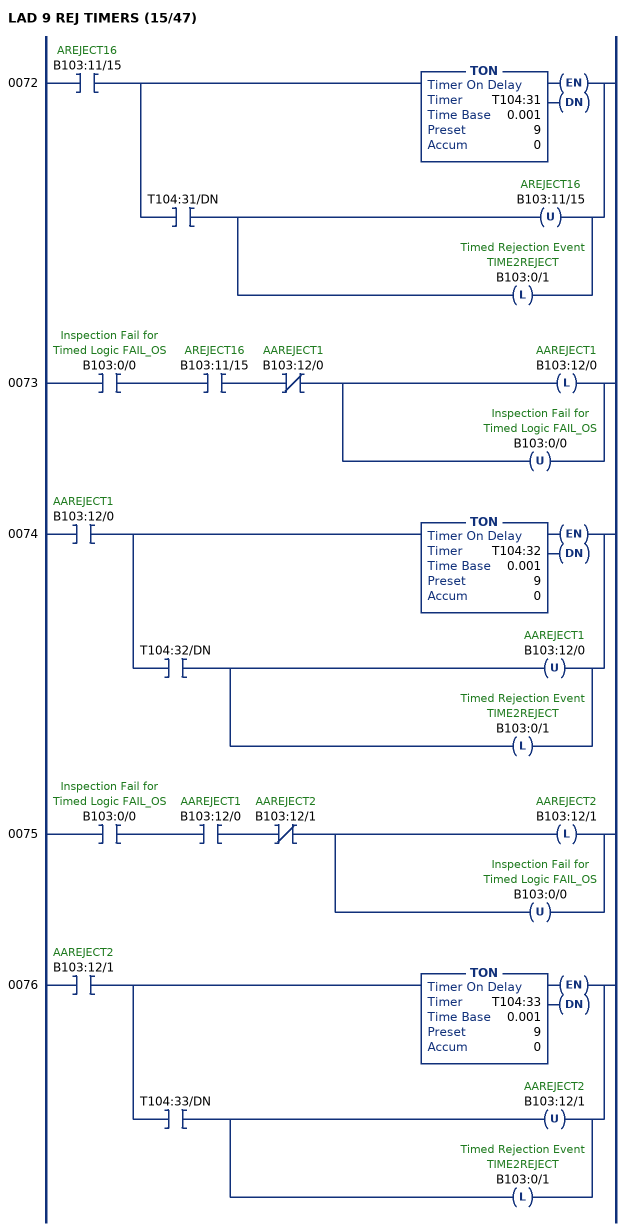
% Rung: 72 %
SOR XIC B103:11/15 BST TON T104:31 0.001 9 0 NXB XIC T104:31/DN BST OTU B103:11/15 NXB OTL B103:0/1 BND BND EOR
%   B103:11/15  AREJECT16 %
%   B103:0/1  TIME2REJECT  "Timed Rejection Event" %
% Rung: 73 %
SOR XIC B103:0/0 XIC B103:11/15 XIO B103:12/0 BST OTL B103:12/0 NXB OTU B103:0/0 BND EOR
%   B103:0/0  FAIL_OS  "Inspection Fail for Timed Logic" %
%   B103:11/15  AREJECT16 %
%   B103:12/0  AAREJECT1 %
% Rung: 74 %
SOR XIC B103:12/0 BST TON T104:32 0.001 9 0 NXB XIC T104:32/DN BST OTU B103:12/0 NXB OTL B103:0/1 BND BND EOR
%   B103:12/0  AAREJECT1 %
%   B103:0/1  TIME2REJECT  "Timed Rejection Event" %
% Rung: 75 %
SOR XIC B103:0/0 XIC B103:12/0 XIO B103:12/1 BST OTL B103:12/1 NXB OTU B103:0/0 BND EOR
%   B103:0/0  FAIL_OS  "Inspection Fail for Timed Logic" %
%   B103:12/0  AAREJECT1 %
%   B103:12/1  AAREJECT2 %
% Rung: 76 %
SOR XIC B103:12/1 BST TON T104:33 0.001 9 0 NXB XIC T104:33/DN BST OTU B103:12/1 NXB OTL B103:0/1 BND BND EOR
%   B103:12/1  AAREJECT2 %
%   B103:0/1  TIME2REJECT  "Timed Rejection Event" %

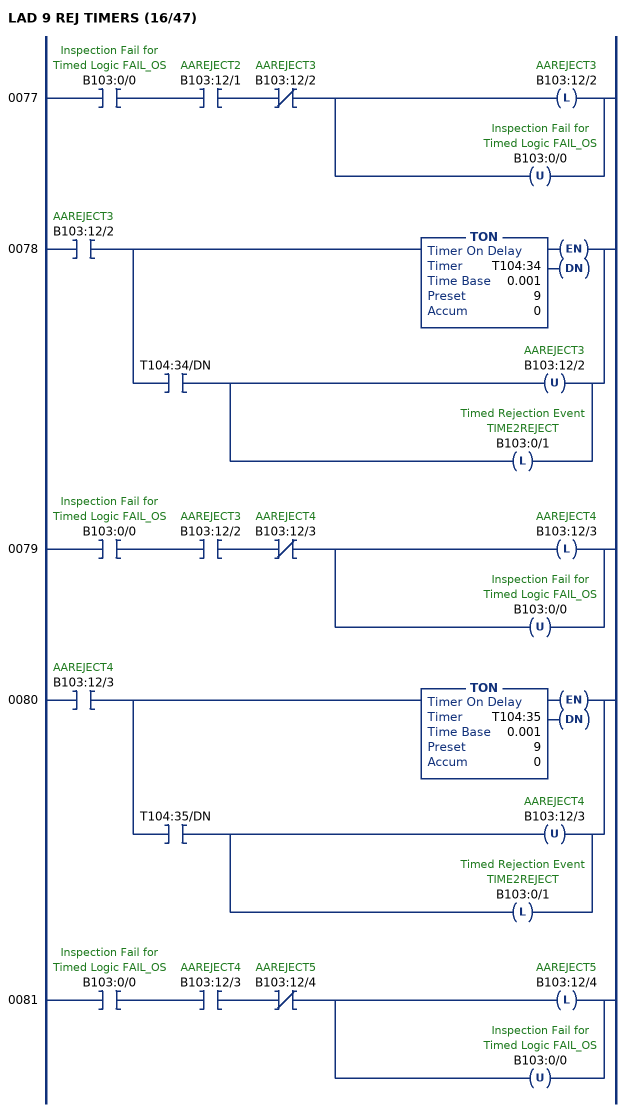
% Rung: 77 %
SOR XIC B103:0/0 XIC B103:12/1 XIO B103:12/2 BST OTL B103:12/2 NXB OTU B103:0/0 BND EOR
%   B103:0/0  FAIL_OS  "Inspection Fail for Timed Logic" %
%   B103:12/1  AAREJECT2 %
%   B103:12/2  AAREJECT3 %
% Rung: 78 %
SOR XIC B103:12/2 BST TON T104:34 0.001 9 0 NXB XIC T104:34/DN BST OTU B103:12/2 NXB OTL B103:0/1 BND BND EOR
%   B103:12/2  AAREJECT3 %
%   B103:0/1  TIME2REJECT  "Timed Rejection Event" %
% Rung: 79 %
SOR XIC B103:0/0 XIC B103:12/2 XIO B103:12/3 BST OTL B103:12/3 NXB OTU B103:0/0 BND EOR
%   B103:0/0  FAIL_OS  "Inspection Fail for Timed Logic" %
%   B103:12/2  AAREJECT3 %
%   B103:12/3  AAREJECT4 %
% Rung: 80 %
SOR XIC B103:12/3 BST TON T104:35 0.001 9 0 NXB XIC T104:35/DN BST OTU B103:12/3 NXB OTL B103:0/1 BND BND EOR
%   B103:12/3  AAREJECT4 %
%   B103:0/1  TIME2REJECT  "Timed Rejection Event" %
% Rung: 81 %
SOR XIC B103:0/0 XIC B103:12/3 XIO B103:12/4 BST OTL B103:12/4 NXB OTU B103:0/0 BND EOR
%   B103:0/0  FAIL_OS  "Inspection Fail for Timed Logic" %
%   B103:12/3  AAREJECT4 %
%   B103:12/4  AAREJECT5 %

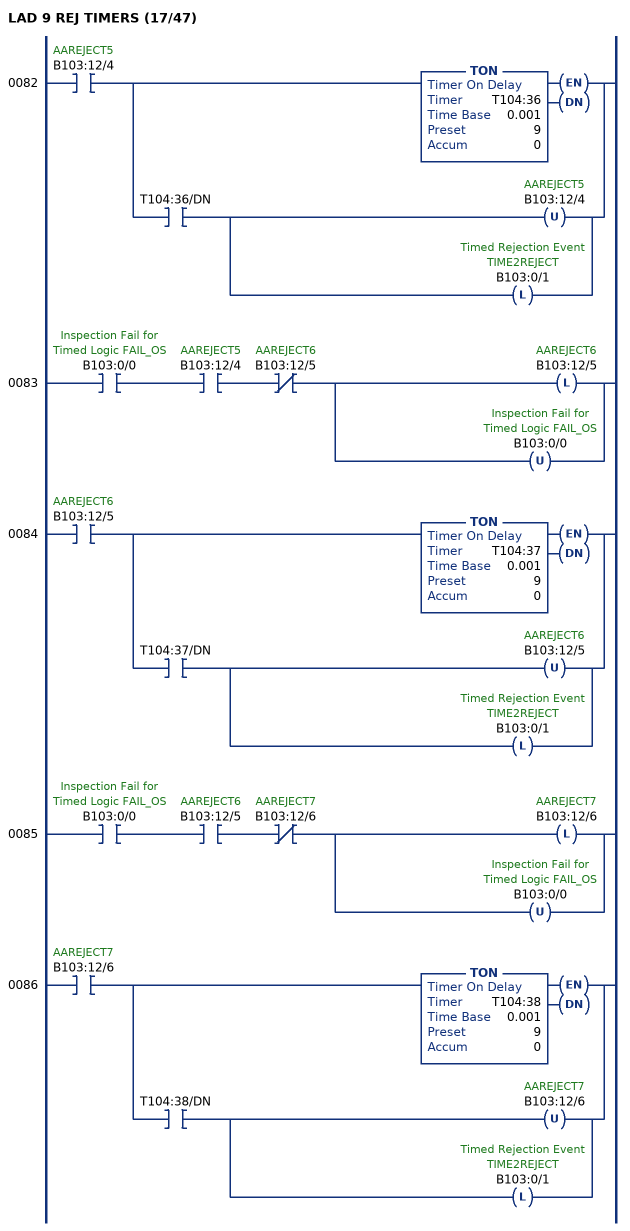
% Rung: 82 %
SOR XIC B103:12/4 BST TON T104:36 0.001 9 0 NXB XIC T104:36/DN BST OTU B103:12/4 NXB OTL B103:0/1 BND BND EOR
%   B103:12/4  AAREJECT5 %
%   B103:0/1  TIME2REJECT  "Timed Rejection Event" %
% Rung: 83 %
SOR XIC B103:0/0 XIC B103:12/4 XIO B103:12/5 BST OTL B103:12/5 NXB OTU B103:0/0 BND EOR
%   B103:0/0  FAIL_OS  "Inspection Fail for Timed Logic" %
%   B103:12/4  AAREJECT5 %
%   B103:12/5  AAREJECT6 %
% Rung: 84 %
SOR XIC B103:12/5 BST TON T104:37 0.001 9 0 NXB XIC T104:37/DN BST OTU B103:12/5 NXB OTL B103:0/1 BND BND EOR
%   B103:12/5  AAREJECT6 %
%   B103:0/1  TIME2REJECT  "Timed Rejection Event" %
% Rung: 85 %
SOR XIC B103:0/0 XIC B103:12/5 XIO B103:12/6 BST OTL B103:12/6 NXB OTU B103:0/0 BND EOR
%   B103:0/0  FAIL_OS  "Inspection Fail for Timed Logic" %
%   B103:12/5  AAREJECT6 %
%   B103:12/6  AAREJECT7 %
% Rung: 86 %
SOR XIC B103:12/6 BST TON T104:38 0.001 9 0 NXB XIC T104:38/DN BST OTU B103:12/6 NXB OTL B103:0/1 BND BND EOR
%   B103:12/6  AAREJECT7 %
%   B103:0/1  TIME2REJECT  "Timed Rejection Event" %

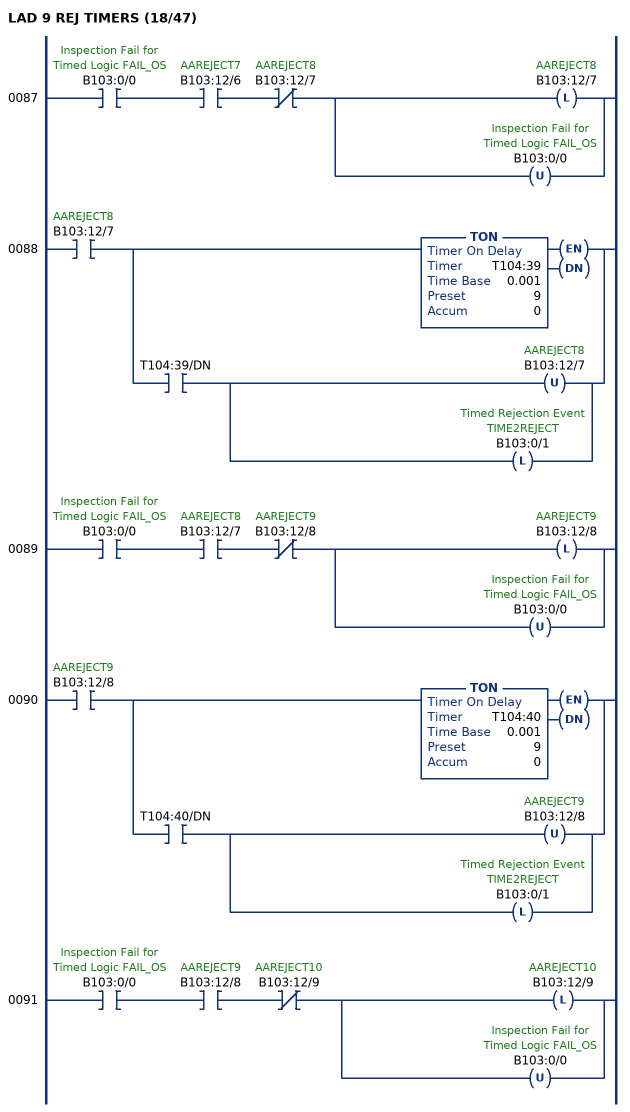
% Rung: 87 %
SOR XIC B103:0/0 XIC B103:12/6 XIO B103:12/7 BST OTL B103:12/7 NXB OTU B103:0/0 BND EOR
%   B103:0/0  FAIL_OS  "Inspection Fail for Timed Logic" %
%   B103:12/6  AAREJECT7 %
%   B103:12/7  AAREJECT8 %
% Rung: 88 %
SOR XIC B103:12/7 BST TON T104:39 0.001 9 0 NXB XIC T104:39/DN BST OTU B103:12/7 NXB OTL B103:0/1 BND BND EOR
%   B103:12/7  AAREJECT8 %
%   B103:0/1  TIME2REJECT  "Timed Rejection Event" %
% Rung: 89 %
SOR XIC B103:0/0 XIC B103:12/7 XIO B103:12/8 BST OTL B103:12/8 NXB OTU B103:0/0 BND EOR
%   B103:0/0  FAIL_OS  "Inspection Fail for Timed Logic" %
%   B103:12/7  AAREJECT8 %
%   B103:12/8  AAREJECT9 %
% Rung: 90 %
SOR XIC B103:12/8 BST TON T104:40 0.001 9 0 NXB XIC T104:40/DN BST OTU B103:12/8 NXB OTL B103:0/1 BND BND EOR
%   B103:12/8  AAREJECT9 %
%   B103:0/1  TIME2REJECT  "Timed Rejection Event" %
% Rung: 91 %
SOR XIC B103:0/0 XIC B103:12/8 XIO B103:12/9 BST OTL B103:12/9 NXB OTU B103:0/0 BND EOR
%   B103:0/0  FAIL_OS  "Inspection Fail for Timed Logic" %
%   B103:12/8  AAREJECT9 %
%   B103:12/9  AAREJECT10 %

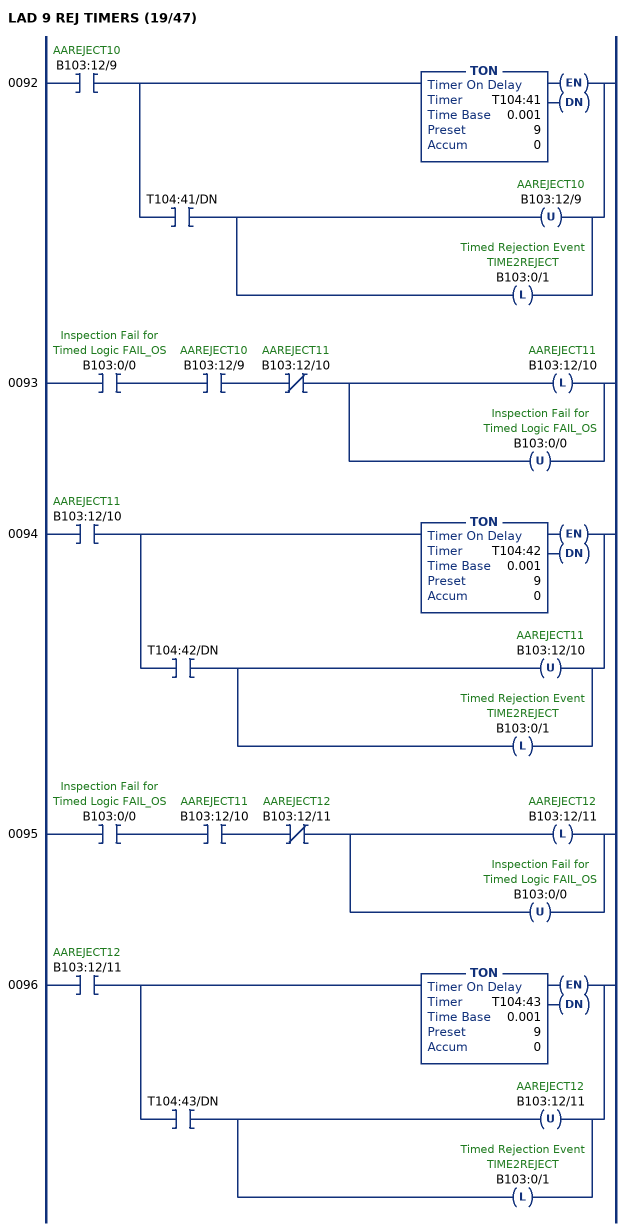
% Rung: 92 %
SOR XIC B103:12/9 BST TON T104:41 0.001 9 0 NXB XIC T104:41/DN BST OTU B103:12/9 NXB OTL B103:0/1 BND BND EOR
%   B103:12/9  AAREJECT10 %
%   B103:0/1  TIME2REJECT  "Timed Rejection Event" %
% Rung: 93 %
SOR XIC B103:0/0 XIC B103:12/9 XIO B103:12/10 BST OTL B103:12/10 NXB OTU B103:0/0 BND EOR
%   B103:0/0  FAIL_OS  "Inspection Fail for Timed Logic" %
%   B103:12/9  AAREJECT10 %
%   B103:12/10  AAREJECT11 %
% Rung: 94 %
SOR XIC B103:12/10 BST TON T104:42 0.001 9 0 NXB XIC T104:42/DN BST OTU B103:12/10 NXB OTL B103:0/1 BND BND EOR
%   B103:12/10  AAREJECT11 %
%   B103:0/1  TIME2REJECT  "Timed Rejection Event" %
% Rung: 95 %
SOR XIC B103:0/0 XIC B103:12/10 XIO B103:12/11 BST OTL B103:12/11 NXB OTU B103:0/0 BND EOR
%   B103:0/0  FAIL_OS  "Inspection Fail for Timed Logic" %
%   B103:12/10  AAREJECT11 %
%   B103:12/11  AAREJECT12 %
% Rung: 96 %
SOR XIC B103:12/11 BST TON T104:43 0.001 9 0 NXB XIC T104:43/DN BST OTU B103:12/11 NXB OTL B103:0/1 BND BND EOR
%   B103:12/11  AAREJECT12 %
%   B103:0/1  TIME2REJECT  "Timed Rejection Event" %

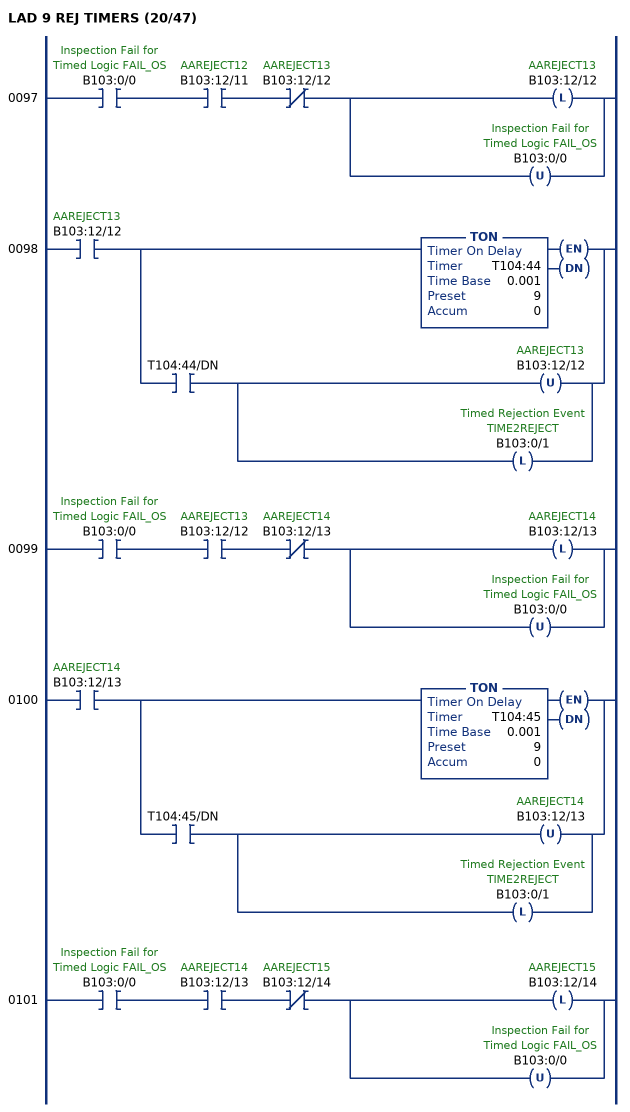
% Rung: 97 %
SOR XIC B103:0/0 XIC B103:12/11 XIO B103:12/12 BST OTL B103:12/12 NXB OTU B103:0/0 BND EOR
%   B103:0/0  FAIL_OS  "Inspection Fail for Timed Logic" %
%   B103:12/11  AAREJECT12 %
%   B103:12/12  AAREJECT13 %
% Rung: 98 %
SOR XIC B103:12/12 BST TON T104:44 0.001 9 0 NXB XIC T104:44/DN BST OTU B103:12/12 NXB OTL B103:0/1 BND BND EOR
%   B103:12/12  AAREJECT13 %
%   B103:0/1  TIME2REJECT  "Timed Rejection Event" %
% Rung: 99 %
SOR XIC B103:0/0 XIC B103:12/12 XIO B103:12/13 BST OTL B103:12/13 NXB OTU B103:0/0 BND EOR
%   B103:0/0  FAIL_OS  "Inspection Fail for Timed Logic" %
%   B103:12/12  AAREJECT13 %
%   B103:12/13  AAREJECT14 %
% Rung: 100 %
SOR XIC B103:12/13 BST TON T104:45 0.001 9 0 NXB XIC T104:45/DN BST OTU B103:12/13 NXB OTL B103:0/1 BND BND EOR
%   B103:12/13  AAREJECT14 %
%   B103:0/1  TIME2REJECT  "Timed Rejection Event" %
% Rung: 101 %
SOR XIC B103:0/0 XIC B103:12/13 XIO B103:12/14 BST OTL B103:12/14 NXB OTU B103:0/0 BND EOR
%   B103:0/0  FAIL_OS  "Inspection Fail for Timed Logic" %
%   B103:12/13  AAREJECT14 %
%   B103:12/14  AAREJECT15 %

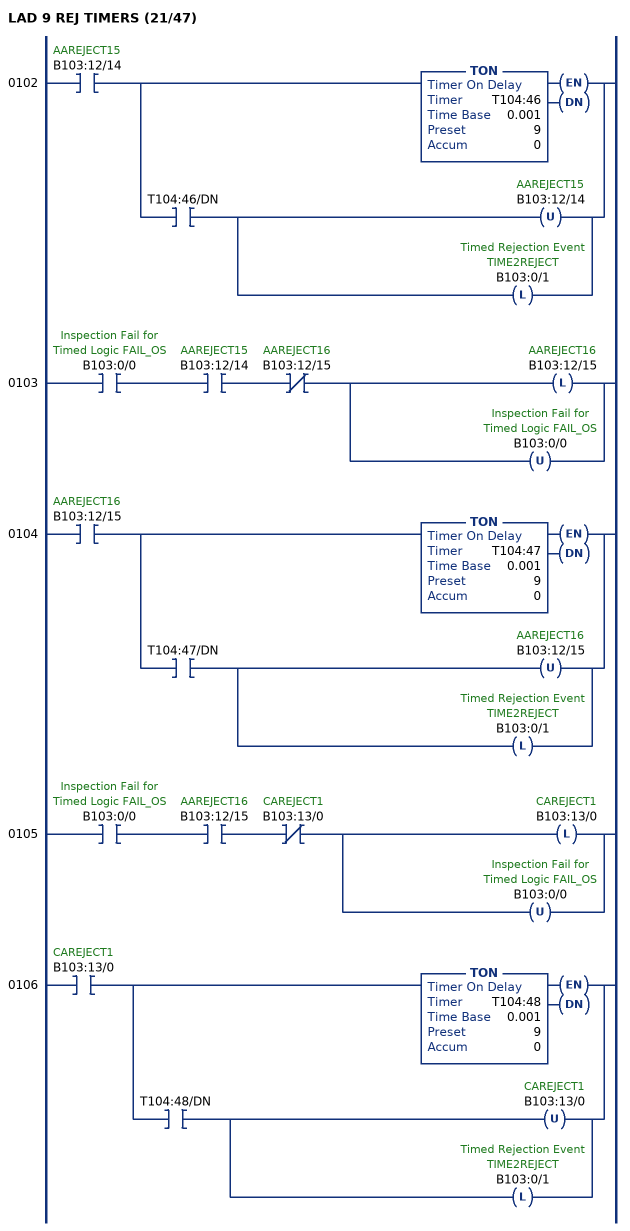
% Rung: 102 %
SOR XIC B103:12/14 BST TON T104:46 0.001 9 0 NXB XIC T104:46/DN BST OTU B103:12/14 NXB OTL B103:0/1 BND BND EOR
%   B103:12/14  AAREJECT15 %
%   B103:0/1  TIME2REJECT  "Timed Rejection Event" %
% Rung: 103 %
SOR XIC B103:0/0 XIC B103:12/14 XIO B103:12/15 BST OTL B103:12/15 NXB OTU B103:0/0 BND EOR
%   B103:0/0  FAIL_OS  "Inspection Fail for Timed Logic" %
%   B103:12/14  AAREJECT15 %
%   B103:12/15  AAREJECT16 %
% Rung: 104 %
SOR XIC B103:12/15 BST TON T104:47 0.001 9 0 NXB XIC T104:47/DN BST OTU B103:12/15 NXB OTL B103:0/1 BND BND EOR
%   B103:12/15  AAREJECT16 %
%   B103:0/1  TIME2REJECT  "Timed Rejection Event" %
% Rung: 105 %
SOR XIC B103:0/0 XIC B103:12/15 XIO B103:13/0 BST OTL B103:13/0 NXB OTU B103:0/0 BND EOR
%   B103:0/0  FAIL_OS  "Inspection Fail for Timed Logic" %
%   B103:12/15  AAREJECT16 %
%   B103:13/0  CAREJECT1 %
% Rung: 106 %
SOR XIC B103:13/0 BST TON T104:48 0.001 9 0 NXB XIC T104:48/DN BST OTU B103:13/0 NXB OTL B103:0/1 BND BND EOR
%   B103:13/0  CAREJECT1 %
%   B103:0/1  TIME2REJECT  "Timed Rejection Event" %

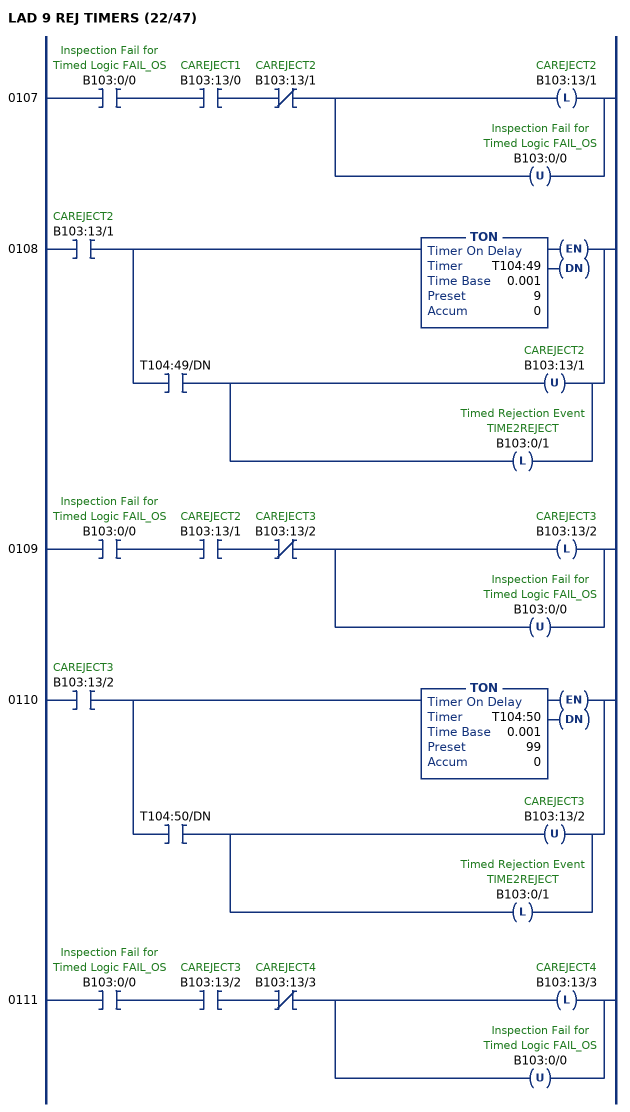
% Rung: 107 %
SOR XIC B103:0/0 XIC B103:13/0 XIO B103:13/1 BST OTL B103:13/1 NXB OTU B103:0/0 BND EOR
%   B103:0/0  FAIL_OS  "Inspection Fail for Timed Logic" %
%   B103:13/0  CAREJECT1 %
%   B103:13/1  CAREJECT2 %
% Rung: 108 %
SOR XIC B103:13/1 BST TON T104:49 0.001 9 0 NXB XIC T104:49/DN BST OTU B103:13/1 NXB OTL B103:0/1 BND BND EOR
%   B103:13/1  CAREJECT2 %
%   B103:0/1  TIME2REJECT  "Timed Rejection Event" %
% Rung: 109 %
SOR XIC B103:0/0 XIC B103:13/1 XIO B103:13/2 BST OTL B103:13/2 NXB OTU B103:0/0 BND EOR
%   B103:0/0  FAIL_OS  "Inspection Fail for Timed Logic" %
%   B103:13/1  CAREJECT2 %
%   B103:13/2  CAREJECT3 %
% Rung: 110 %
SOR XIC B103:13/2 BST TON T104:50 0.001 99 0 NXB XIC T104:50/DN BST OTU B103:13/2 NXB OTL B103:0/1 BND BND EOR
%   B103:13/2  CAREJECT3 %
%   B103:0/1  TIME2REJECT  "Timed Rejection Event" %
% Rung: 111 %
SOR XIC B103:0/0 XIC B103:13/2 XIO B103:13/3 BST OTL B103:13/3 NXB OTU B103:0/0 BND EOR
%   B103:0/0  FAIL_OS  "Inspection Fail for Timed Logic" %
%   B103:13/2  CAREJECT3 %
%   B103:13/3  CAREJECT4 %

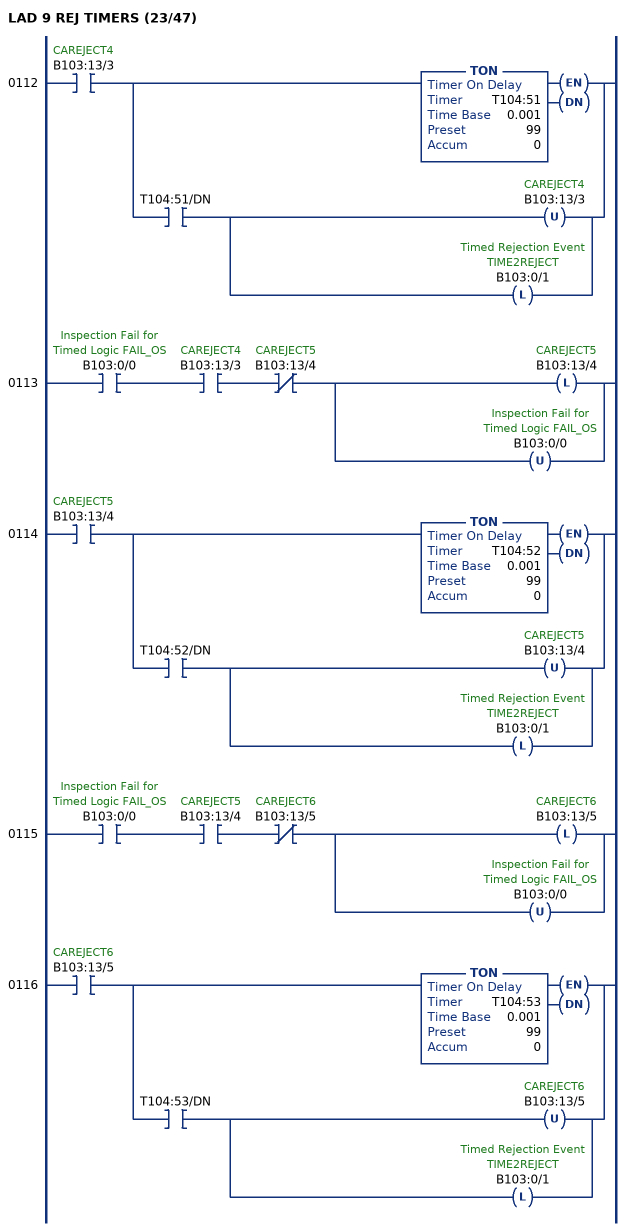
% Rung: 112 %
SOR XIC B103:13/3 BST TON T104:51 0.001 99 0 NXB XIC T104:51/DN BST OTU B103:13/3 NXB OTL B103:0/1 BND BND EOR
%   B103:13/3  CAREJECT4 %
%   B103:0/1  TIME2REJECT  "Timed Rejection Event" %
% Rung: 113 %
SOR XIC B103:0/0 XIC B103:13/3 XIO B103:13/4 BST OTL B103:13/4 NXB OTU B103:0/0 BND EOR
%   B103:0/0  FAIL_OS  "Inspection Fail for Timed Logic" %
%   B103:13/3  CAREJECT4 %
%   B103:13/4  CAREJECT5 %
% Rung: 114 %
SOR XIC B103:13/4 BST TON T104:52 0.001 99 0 NXB XIC T104:52/DN BST OTU B103:13/4 NXB OTL B103:0/1 BND BND EOR
%   B103:13/4  CAREJECT5 %
%   B103:0/1  TIME2REJECT  "Timed Rejection Event" %
% Rung: 115 %
SOR XIC B103:0/0 XIC B103:13/4 XIO B103:13/5 BST OTL B103:13/5 NXB OTU B103:0/0 BND EOR
%   B103:0/0  FAIL_OS  "Inspection Fail for Timed Logic" %
%   B103:13/4  CAREJECT5 %
%   B103:13/5  CAREJECT6 %
% Rung: 116 %
SOR XIC B103:13/5 BST TON T104:53 0.001 99 0 NXB XIC T104:53/DN BST OTU B103:13/5 NXB OTL B103:0/1 BND BND EOR
%   B103:13/5  CAREJECT6 %
%   B103:0/1  TIME2REJECT  "Timed Rejection Event" %

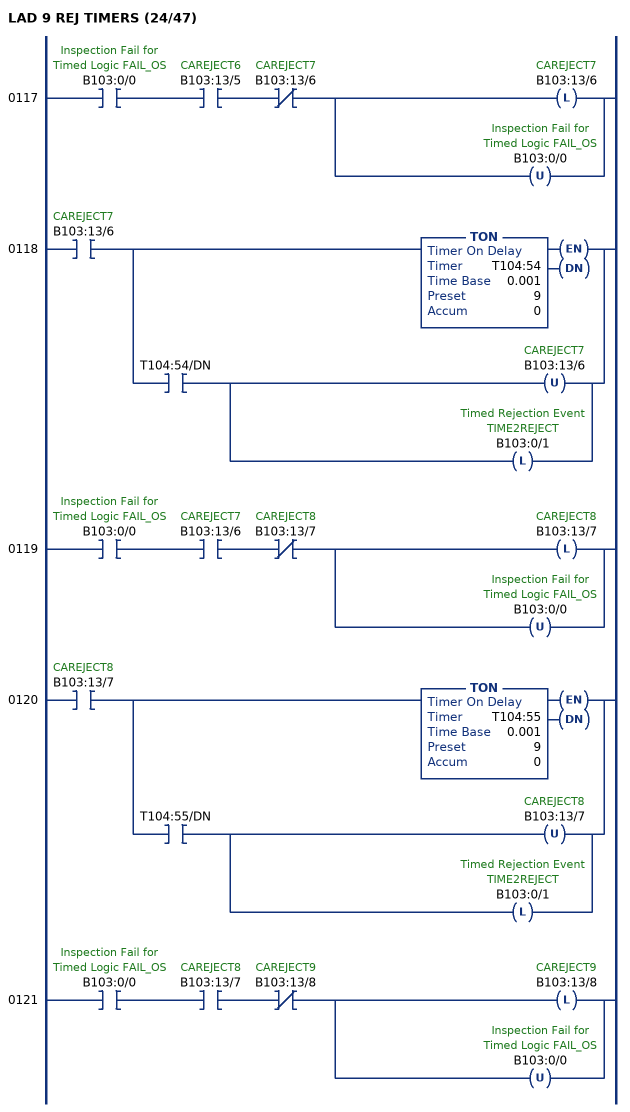
% Rung: 117 %
SOR XIC B103:0/0 XIC B103:13/5 XIO B103:13/6 BST OTL B103:13/6 NXB OTU B103:0/0 BND EOR
%   B103:0/0  FAIL_OS  "Inspection Fail for Timed Logic" %
%   B103:13/5  CAREJECT6 %
%   B103:13/6  CAREJECT7 %
% Rung: 118 %
SOR XIC B103:13/6 BST TON T104:54 0.001 9 0 NXB XIC T104:54/DN BST OTU B103:13/6 NXB OTL B103:0/1 BND BND EOR
%   B103:13/6  CAREJECT7 %
%   B103:0/1  TIME2REJECT  "Timed Rejection Event" %
% Rung: 119 %
SOR XIC B103:0/0 XIC B103:13/6 XIO B103:13/7 BST OTL B103:13/7 NXB OTU B103:0/0 BND EOR
%   B103:0/0  FAIL_OS  "Inspection Fail for Timed Logic" %
%   B103:13/6  CAREJECT7 %
%   B103:13/7  CAREJECT8 %
% Rung: 120 %
SOR XIC B103:13/7 BST TON T104:55 0.001 9 0 NXB XIC T104:55/DN BST OTU B103:13/7 NXB OTL B103:0/1 BND BND EOR
%   B103:13/7  CAREJECT8 %
%   B103:0/1  TIME2REJECT  "Timed Rejection Event" %
% Rung: 121 %
SOR XIC B103:0/0 XIC B103:13/7 XIO B103:13/8 BST OTL B103:13/8 NXB OTU B103:0/0 BND EOR
%   B103:0/0  FAIL_OS  "Inspection Fail for Timed Logic" %
%   B103:13/7  CAREJECT8 %
%   B103:13/8  CAREJECT9 %

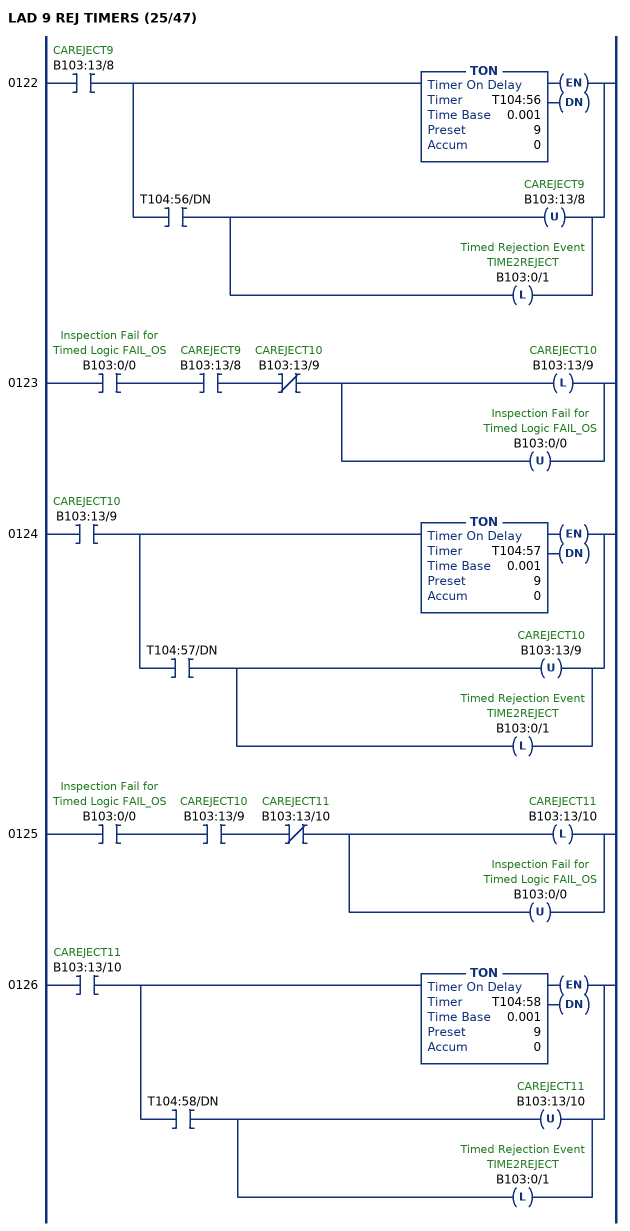
% Rung: 122 %
SOR XIC B103:13/8 BST TON T104:56 0.001 9 0 NXB XIC T104:56/DN BST OTU B103:13/8 NXB OTL B103:0/1 BND BND EOR
%   B103:13/8  CAREJECT9 %
%   B103:0/1  TIME2REJECT  "Timed Rejection Event" %
% Rung: 123 %
SOR XIC B103:0/0 XIC B103:13/8 XIO B103:13/9 BST OTL B103:13/9 NXB OTU B103:0/0 BND EOR
%   B103:0/0  FAIL_OS  "Inspection Fail for Timed Logic" %
%   B103:13/8  CAREJECT9 %
%   B103:13/9  CAREJECT10 %
% Rung: 124 %
SOR XIC B103:13/9 BST TON T104:57 0.001 9 0 NXB XIC T104:57/DN BST OTU B103:13/9 NXB OTL B103:0/1 BND BND EOR
%   B103:13/9  CAREJECT10 %
%   B103:0/1  TIME2REJECT  "Timed Rejection Event" %
% Rung: 125 %
SOR XIC B103:0/0 XIC B103:13/9 XIO B103:13/10 BST OTL B103:13/10 NXB OTU B103:0/0 BND EOR
%   B103:0/0  FAIL_OS  "Inspection Fail for Timed Logic" %
%   B103:13/9  CAREJECT10 %
%   B103:13/10  CAREJECT11 %
% Rung: 126 %
SOR XIC B103:13/10 BST TON T104:58 0.001 9 0 NXB XIC T104:58/DN BST OTU B103:13/10 NXB OTL B103:0/1 BND BND EOR
%   B103:13/10  CAREJECT11 %
%   B103:0/1  TIME2REJECT  "Timed Rejection Event" %

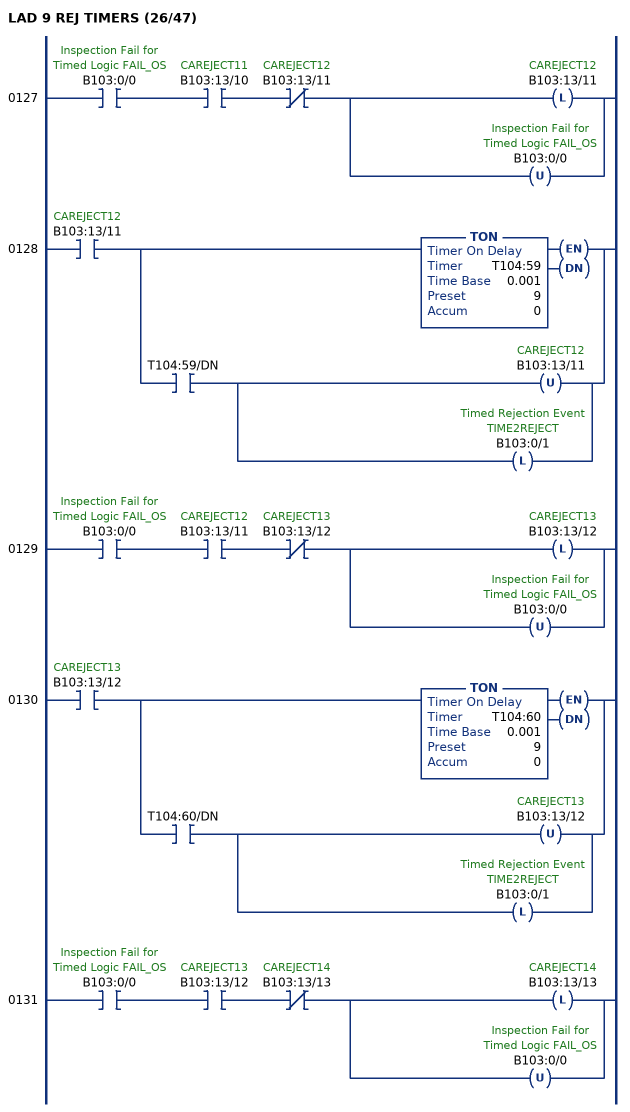
% Rung: 127 %
SOR XIC B103:0/0 XIC B103:13/10 XIO B103:13/11 BST OTL B103:13/11 NXB OTU B103:0/0 BND EOR
%   B103:0/0  FAIL_OS  "Inspection Fail for Timed Logic" %
%   B103:13/10  CAREJECT11 %
%   B103:13/11  CAREJECT12 %
% Rung: 128 %
SOR XIC B103:13/11 BST TON T104:59 0.001 9 0 NXB XIC T104:59/DN BST OTU B103:13/11 NXB OTL B103:0/1 BND BND EOR
%   B103:13/11  CAREJECT12 %
%   B103:0/1  TIME2REJECT  "Timed Rejection Event" %
% Rung: 129 %
SOR XIC B103:0/0 XIC B103:13/11 XIO B103:13/12 BST OTL B103:13/12 NXB OTU B103:0/0 BND EOR
%   B103:0/0  FAIL_OS  "Inspection Fail for Timed Logic" %
%   B103:13/11  CAREJECT12 %
%   B103:13/12  CAREJECT13 %
% Rung: 130 %
SOR XIC B103:13/12 BST TON T104:60 0.001 9 0 NXB XIC T104:60/DN BST OTU B103:13/12 NXB OTL B103:0/1 BND BND EOR
%   B103:13/12  CAREJECT13 %
%   B103:0/1  TIME2REJECT  "Timed Rejection Event" %
% Rung: 131 %
SOR XIC B103:0/0 XIC B103:13/12 XIO B103:13/13 BST OTL B103:13/13 NXB OTU B103:0/0 BND EOR
%   B103:0/0  FAIL_OS  "Inspection Fail for Timed Logic" %
%   B103:13/12  CAREJECT13 %
%   B103:13/13  CAREJECT14 %

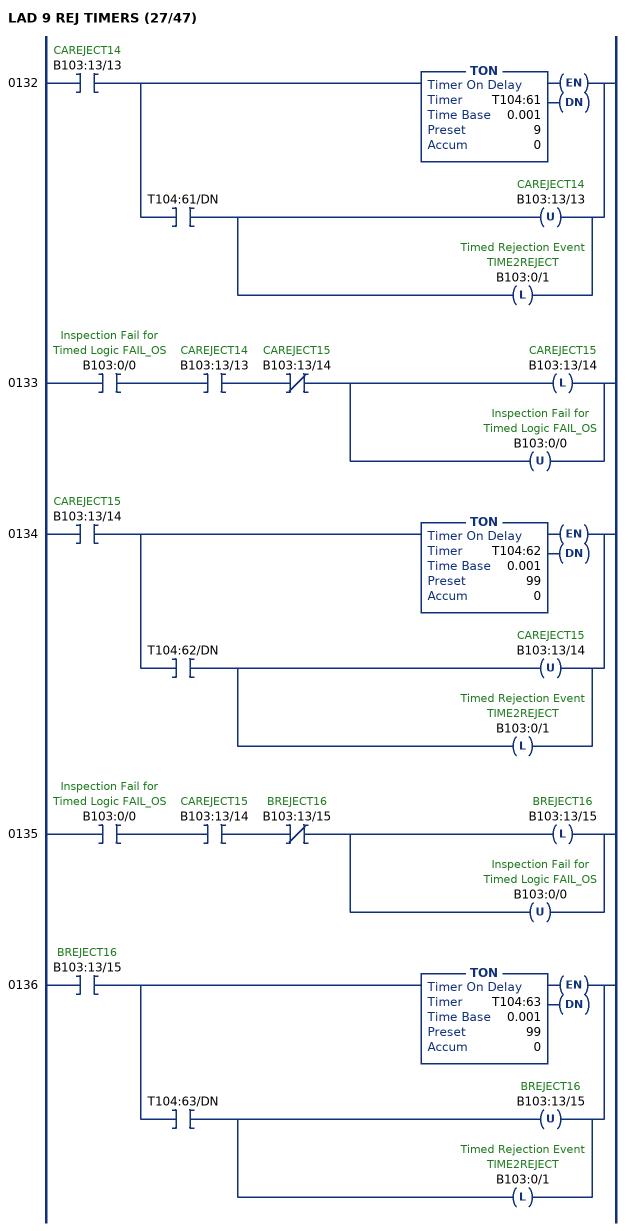
% Rung: 132 %
SOR XIC B103:13/13 BST TON T104:61 0.001 9 0 NXB XIC T104:61/DN BST OTU B103:13/13 NXB OTL B103:0/1 BND BND EOR
%   B103:13/13  CAREJECT14 %
%   B103:0/1  TIME2REJECT  "Timed Rejection Event" %
% Rung: 133 %
SOR XIC B103:0/0 XIC B103:13/13 XIO B103:13/14 BST OTL B103:13/14 NXB OTU B103:0/0 BND EOR
%   B103:0/0  FAIL_OS  "Inspection Fail for Timed Logic" %
%   B103:13/13  CAREJECT14 %
%   B103:13/14  CAREJECT15 %
% Rung: 134 %
SOR XIC B103:13/14 BST TON T104:62 0.001 99 0 NXB XIC T104:62/DN BST OTU B103:13/14 NXB OTL B103:0/1 BND BND EOR
%   B103:13/14  CAREJECT15 %
%   B103:0/1  TIME2REJECT  "Timed Rejection Event" %
% Rung: 135 %
SOR XIC B103:0/0 XIC B103:13/14 XIO B103:13/15 BST OTL B103:13/15 NXB OTU B103:0/0 BND EOR
%   B103:0/0  FAIL_OS  "Inspection Fail for Timed Logic" %
%   B103:13/14  CAREJECT15 %
%   B103:13/15  BREJECT16 %
% Rung: 136 %
SOR XIC B103:13/15 BST TON T104:63 0.001 99 0 NXB XIC T104:63/DN BST OTU B103:13/15 NXB OTL B103:0/1 BND BND EOR
%   B103:13/15  BREJECT16 %
%   B103:0/1  TIME2REJECT  "Timed Rejection Event" %

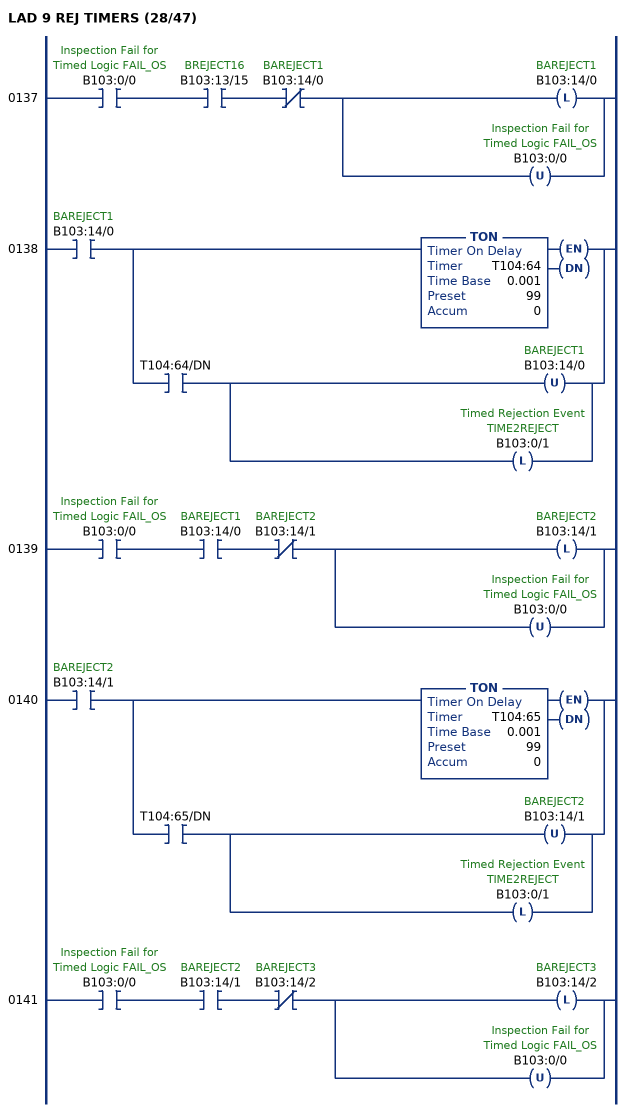
% Rung: 137 %
SOR XIC B103:0/0 XIC B103:13/15 XIO B103:14/0 BST OTL B103:14/0 NXB OTU B103:0/0 BND EOR
%   B103:0/0  FAIL_OS  "Inspection Fail for Timed Logic" %
%   B103:13/15  BREJECT16 %
%   B103:14/0  BAREJECT1 %
% Rung: 138 %
SOR XIC B103:14/0 BST TON T104:64 0.001 99 0 NXB XIC T104:64/DN BST OTU B103:14/0 NXB OTL B103:0/1 BND BND EOR
%   B103:14/0  BAREJECT1 %
%   B103:0/1  TIME2REJECT  "Timed Rejection Event" %
% Rung: 139 %
SOR XIC B103:0/0 XIC B103:14/0 XIO B103:14/1 BST OTL B103:14/1 NXB OTU B103:0/0 BND EOR
%   B103:0/0  FAIL_OS  "Inspection Fail for Timed Logic" %
%   B103:14/0  BAREJECT1 %
%   B103:14/1  BAREJECT2 %
% Rung: 140 %
SOR XIC B103:14/1 BST TON T104:65 0.001 99 0 NXB XIC T104:65/DN BST OTU B103:14/1 NXB OTL B103:0/1 BND BND EOR
%   B103:14/1  BAREJECT2 %
%   B103:0/1  TIME2REJECT  "Timed Rejection Event" %
% Rung: 141 %
SOR XIC B103:0/0 XIC B103:14/1 XIO B103:14/2 BST OTL B103:14/2 NXB OTU B103:0/0 BND EOR
%   B103:0/0  FAIL_OS  "Inspection Fail for Timed Logic" %
%   B103:14/1  BAREJECT2 %
%   B103:14/2  BAREJECT3 %

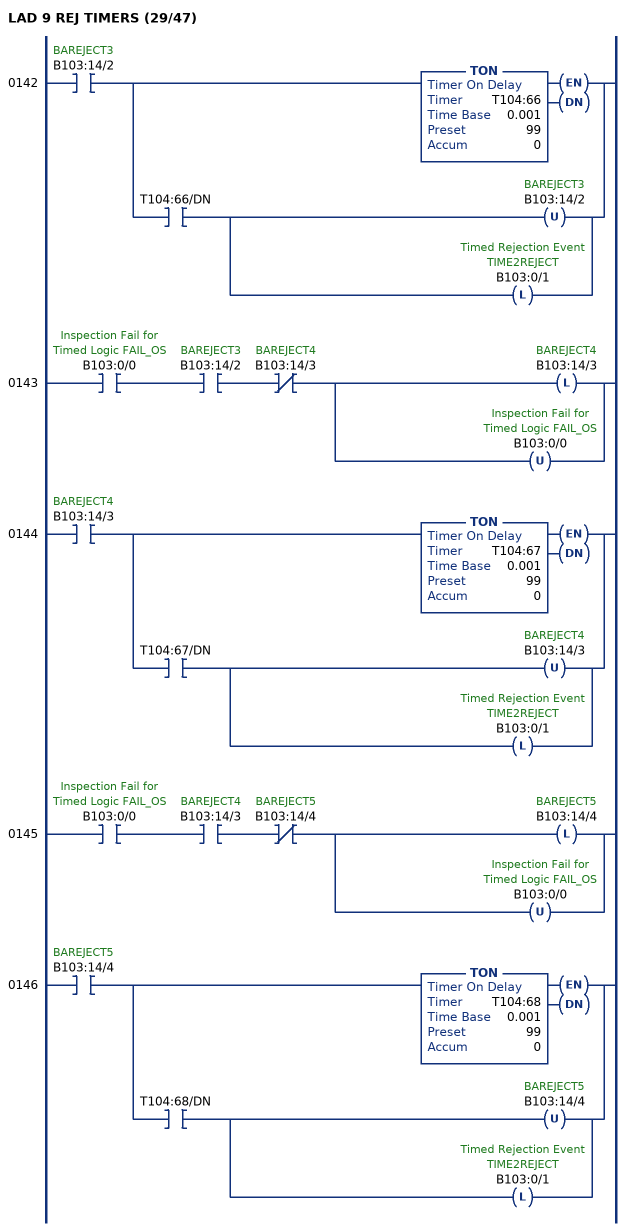
% Rung: 142 %
SOR XIC B103:14/2 BST TON T104:66 0.001 99 0 NXB XIC T104:66/DN BST OTU B103:14/2 NXB OTL B103:0/1 BND BND EOR
%   B103:14/2  BAREJECT3 %
%   B103:0/1  TIME2REJECT  "Timed Rejection Event" %
% Rung: 143 %
SOR XIC B103:0/0 XIC B103:14/2 XIO B103:14/3 BST OTL B103:14/3 NXB OTU B103:0/0 BND EOR
%   B103:0/0  FAIL_OS  "Inspection Fail for Timed Logic" %
%   B103:14/2  BAREJECT3 %
%   B103:14/3  BAREJECT4 %
% Rung: 144 %
SOR XIC B103:14/3 BST TON T104:67 0.001 99 0 NXB XIC T104:67/DN BST OTU B103:14/3 NXB OTL B103:0/1 BND BND EOR
%   B103:14/3  BAREJECT4 %
%   B103:0/1  TIME2REJECT  "Timed Rejection Event" %
% Rung: 145 %
SOR XIC B103:0/0 XIC B103:14/3 XIO B103:14/4 BST OTL B103:14/4 NXB OTU B103:0/0 BND EOR
%   B103:0/0  FAIL_OS  "Inspection Fail for Timed Logic" %
%   B103:14/3  BAREJECT4 %
%   B103:14/4  BAREJECT5 %
% Rung: 146 %
SOR XIC B103:14/4 BST TON T104:68 0.001 99 0 NXB XIC T104:68/DN BST OTU B103:14/4 NXB OTL B103:0/1 BND BND EOR
%   B103:14/4  BAREJECT5 %
%   B103:0/1  TIME2REJECT  "Timed Rejection Event" %

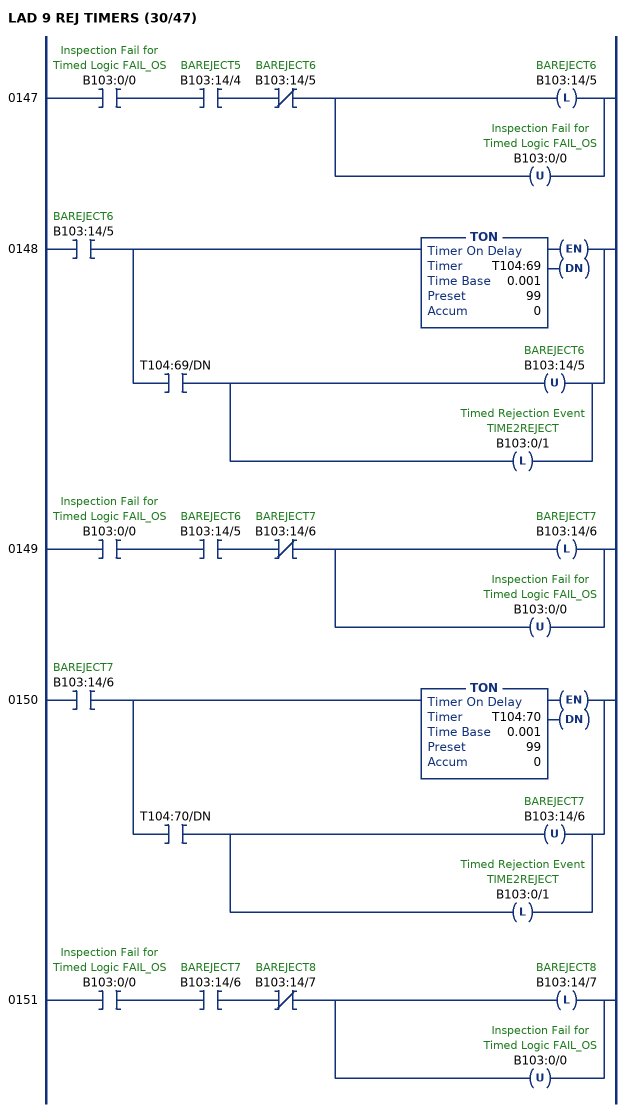
% Rung: 147 %
SOR XIC B103:0/0 XIC B103:14/4 XIO B103:14/5 BST OTL B103:14/5 NXB OTU B103:0/0 BND EOR
%   B103:0/0  FAIL_OS  "Inspection Fail for Timed Logic" %
%   B103:14/4  BAREJECT5 %
%   B103:14/5  BAREJECT6 %
% Rung: 148 %
SOR XIC B103:14/5 BST TON T104:69 0.001 99 0 NXB XIC T104:69/DN BST OTU B103:14/5 NXB OTL B103:0/1 BND BND EOR
%   B103:14/5  BAREJECT6 %
%   B103:0/1  TIME2REJECT  "Timed Rejection Event" %
% Rung: 149 %
SOR XIC B103:0/0 XIC B103:14/5 XIO B103:14/6 BST OTL B103:14/6 NXB OTU B103:0/0 BND EOR
%   B103:0/0  FAIL_OS  "Inspection Fail for Timed Logic" %
%   B103:14/5  BAREJECT6 %
%   B103:14/6  BAREJECT7 %
% Rung: 150 %
SOR XIC B103:14/6 BST TON T104:70 0.001 99 0 NXB XIC T104:70/DN BST OTU B103:14/6 NXB OTL B103:0/1 BND BND EOR
%   B103:14/6  BAREJECT7 %
%   B103:0/1  TIME2REJECT  "Timed Rejection Event" %
% Rung: 151 %
SOR XIC B103:0/0 XIC B103:14/6 XIO B103:14/7 BST OTL B103:14/7 NXB OTU B103:0/0 BND EOR
%   B103:0/0  FAIL_OS  "Inspection Fail for Timed Logic" %
%   B103:14/6  BAREJECT7 %
%   B103:14/7  BAREJECT8 %

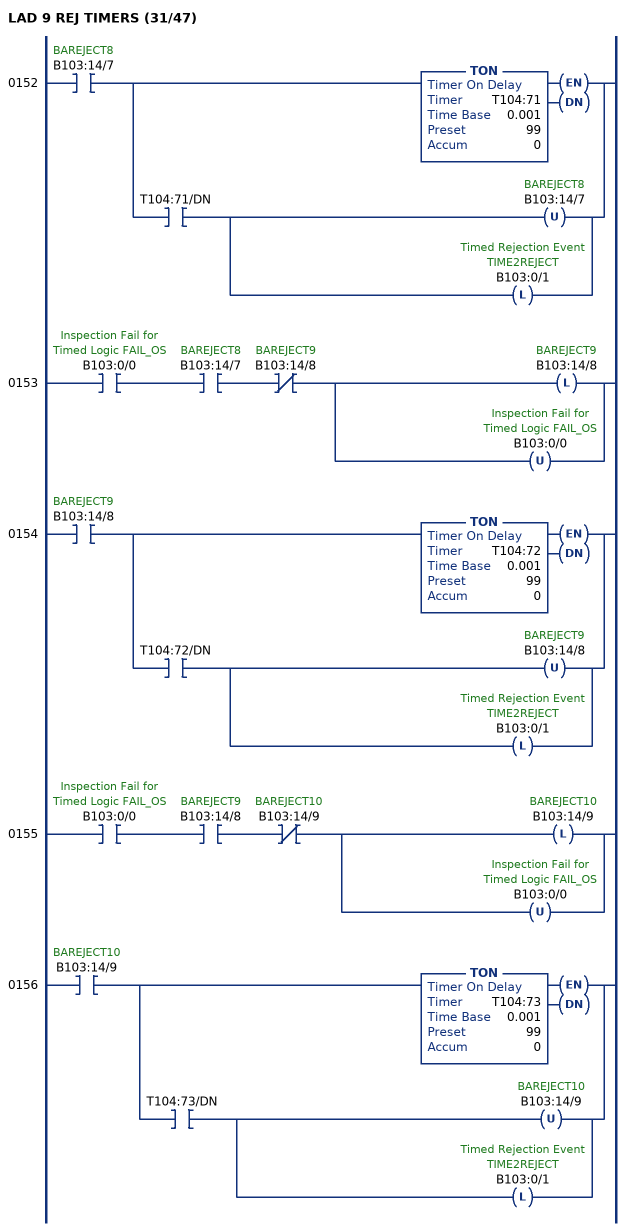
% Rung: 152 %
SOR XIC B103:14/7 BST TON T104:71 0.001 99 0 NXB XIC T104:71/DN BST OTU B103:14/7 NXB OTL B103:0/1 BND BND EOR
%   B103:14/7  BAREJECT8 %
%   B103:0/1  TIME2REJECT  "Timed Rejection Event" %
% Rung: 153 %
SOR XIC B103:0/0 XIC B103:14/7 XIO B103:14/8 BST OTL B103:14/8 NXB OTU B103:0/0 BND EOR
%   B103:0/0  FAIL_OS  "Inspection Fail for Timed Logic" %
%   B103:14/7  BAREJECT8 %
%   B103:14/8  BAREJECT9 %
% Rung: 154 %
SOR XIC B103:14/8 BST TON T104:72 0.001 99 0 NXB XIC T104:72/DN BST OTU B103:14/8 NXB OTL B103:0/1 BND BND EOR
%   B103:14/8  BAREJECT9 %
%   B103:0/1  TIME2REJECT  "Timed Rejection Event" %
% Rung: 155 %
SOR XIC B103:0/0 XIC B103:14/8 XIO B103:14/9 BST OTL B103:14/9 NXB OTU B103:0/0 BND EOR
%   B103:0/0  FAIL_OS  "Inspection Fail for Timed Logic" %
%   B103:14/8  BAREJECT9 %
%   B103:14/9  BAREJECT10 %
% Rung: 156 %
SOR XIC B103:14/9 BST TON T104:73 0.001 99 0 NXB XIC T104:73/DN BST OTU B103:14/9 NXB OTL B103:0/1 BND BND EOR
%   B103:14/9  BAREJECT10 %
%   B103:0/1  TIME2REJECT  "Timed Rejection Event" %

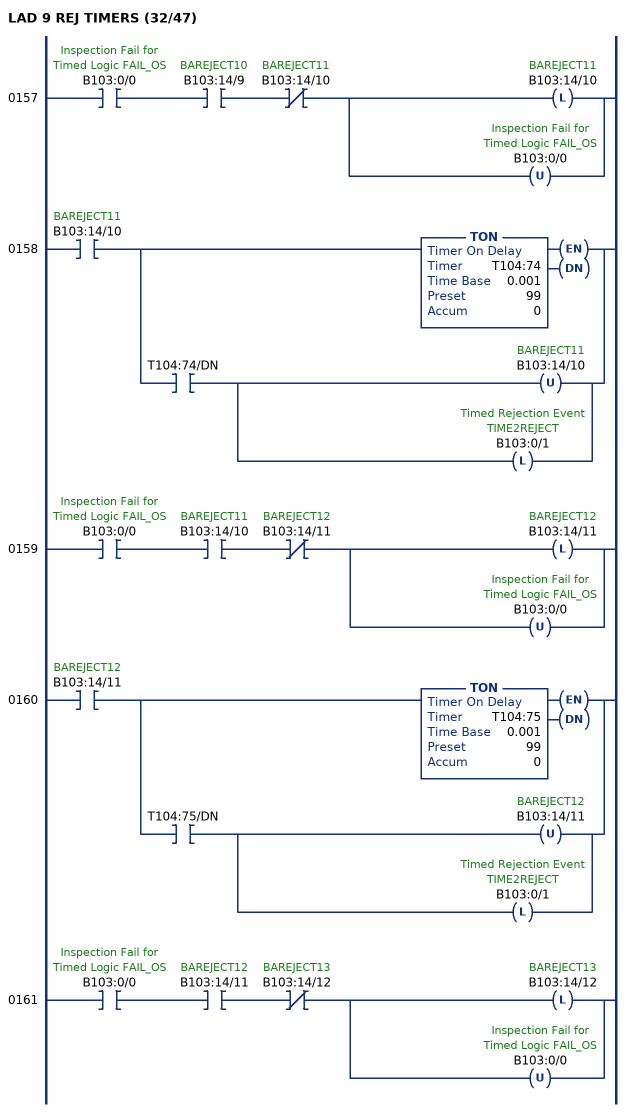
% Rung: 157 %
SOR XIC B103:0/0 XIC B103:14/9 XIO B103:14/10 BST OTL B103:14/10 NXB OTU B103:0/0 BND EOR
%   B103:0/0  FAIL_OS  "Inspection Fail for Timed Logic" %
%   B103:14/9  BAREJECT10 %
%   B103:14/10  BAREJECT11 %
% Rung: 158 %
SOR XIC B103:14/10 BST TON T104:74 0.001 99 0 NXB XIC T104:74/DN BST OTU B103:14/10 NXB OTL B103:0/1 BND BND EOR
%   B103:14/10  BAREJECT11 %
%   B103:0/1  TIME2REJECT  "Timed Rejection Event" %
% Rung: 159 %
SOR XIC B103:0/0 XIC B103:14/10 XIO B103:14/11 BST OTL B103:14/11 NXB OTU B103:0/0 BND EOR
%   B103:0/0  FAIL_OS  "Inspection Fail for Timed Logic" %
%   B103:14/10  BAREJECT11 %
%   B103:14/11  BAREJECT12 %
% Rung: 160 %
SOR XIC B103:14/11 BST TON T104:75 0.001 99 0 NXB XIC T104:75/DN BST OTU B103:14/11 NXB OTL B103:0/1 BND BND EOR
%   B103:14/11  BAREJECT12 %
%   B103:0/1  TIME2REJECT  "Timed Rejection Event" %
% Rung: 161 %
SOR XIC B103:0/0 XIC B103:14/11 XIO B103:14/12 BST OTL B103:14/12 NXB OTU B103:0/0 BND EOR
%   B103:0/0  FAIL_OS  "Inspection Fail for Timed Logic" %
%   B103:14/11  BAREJECT12 %
%   B103:14/12  BAREJECT13 %

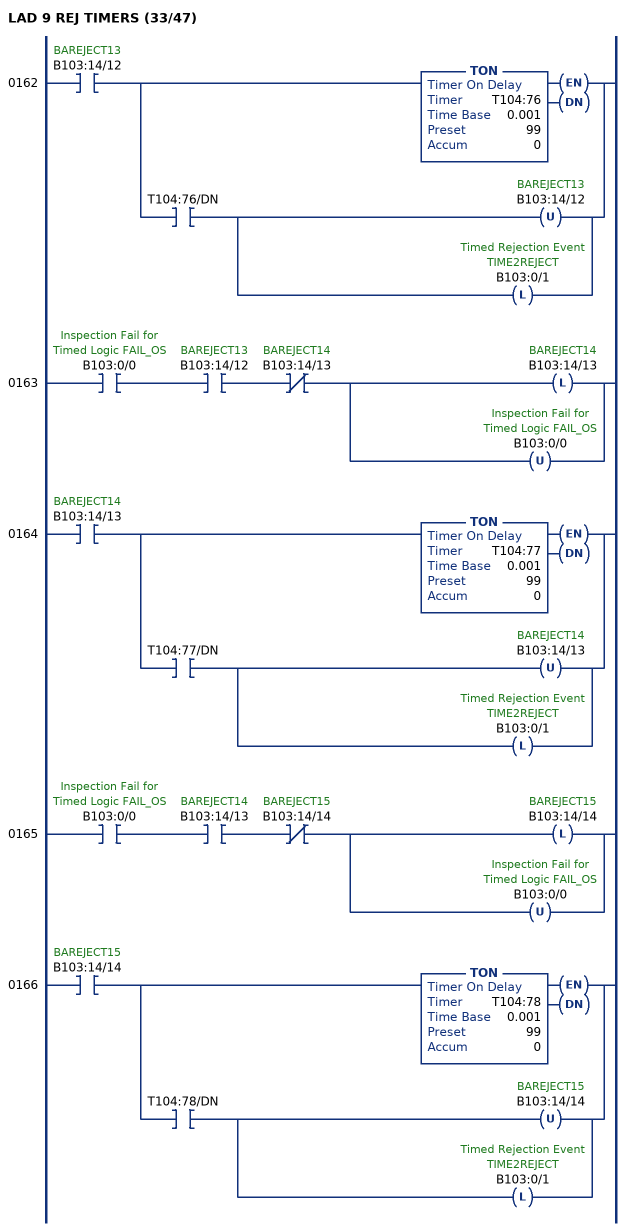
% Rung: 162 %
SOR XIC B103:14/12 BST TON T104:76 0.001 99 0 NXB XIC T104:76/DN BST OTU B103:14/12 NXB OTL B103:0/1 BND BND EOR
%   B103:14/12  BAREJECT13 %
%   B103:0/1  TIME2REJECT  "Timed Rejection Event" %
% Rung: 163 %
SOR XIC B103:0/0 XIC B103:14/12 XIO B103:14/13 BST OTL B103:14/13 NXB OTU B103:0/0 BND EOR
%   B103:0/0  FAIL_OS  "Inspection Fail for Timed Logic" %
%   B103:14/12  BAREJECT13 %
%   B103:14/13  BAREJECT14 %
% Rung: 164 %
SOR XIC B103:14/13 BST TON T104:77 0.001 99 0 NXB XIC T104:77/DN BST OTU B103:14/13 NXB OTL B103:0/1 BND BND EOR
%   B103:14/13  BAREJECT14 %
%   B103:0/1  TIME2REJECT  "Timed Rejection Event" %
% Rung: 165 %
SOR XIC B103:0/0 XIC B103:14/13 XIO B103:14/14 BST OTL B103:14/14 NXB OTU B103:0/0 BND EOR
%   B103:0/0  FAIL_OS  "Inspection Fail for Timed Logic" %
%   B103:14/13  BAREJECT14 %
%   B103:14/14  BAREJECT15 %
% Rung: 166 %
SOR XIC B103:14/14 BST TON T104:78 0.001 99 0 NXB XIC T104:78/DN BST OTU B103:14/14 NXB OTL B103:0/1 BND BND EOR
%   B103:14/14  BAREJECT15 %
%   B103:0/1  TIME2REJECT  "Timed Rejection Event" %

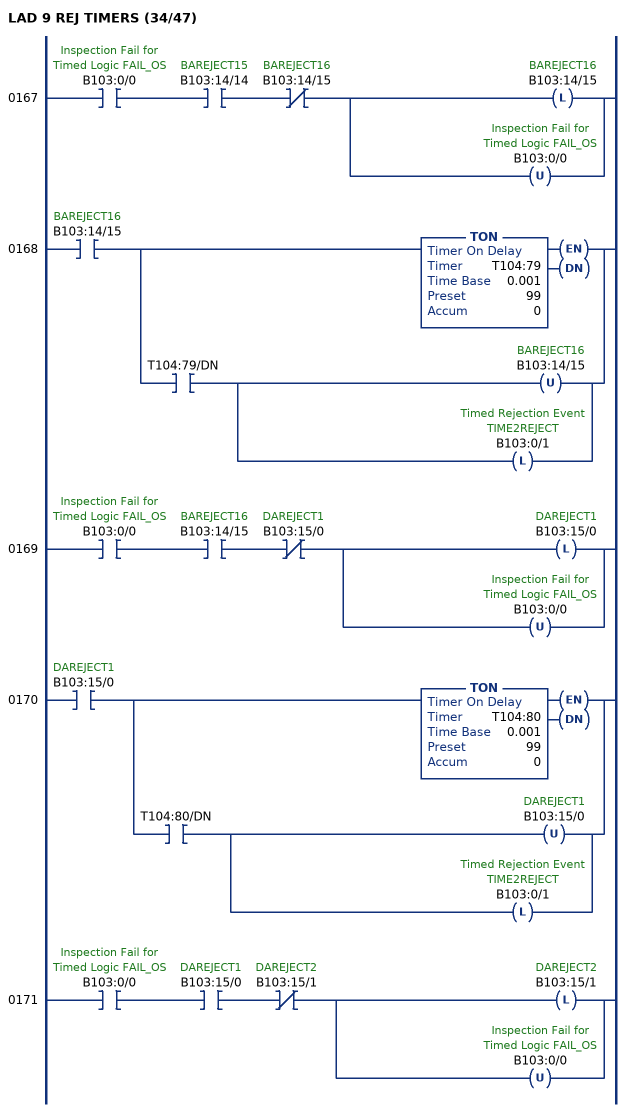
% Rung: 167 %
SOR XIC B103:0/0 XIC B103:14/14 XIO B103:14/15 BST OTL B103:14/15 NXB OTU B103:0/0 BND EOR
%   B103:0/0  FAIL_OS  "Inspection Fail for Timed Logic" %
%   B103:14/14  BAREJECT15 %
%   B103:14/15  BAREJECT16 %
% Rung: 168 %
SOR XIC B103:14/15 BST TON T104:79 0.001 99 0 NXB XIC T104:79/DN BST OTU B103:14/15 NXB OTL B103:0/1 BND BND EOR
%   B103:14/15  BAREJECT16 %
%   B103:0/1  TIME2REJECT  "Timed Rejection Event" %
% Rung: 169 %
SOR XIC B103:0/0 XIC B103:14/15 XIO B103:15/0 BST OTL B103:15/0 NXB OTU B103:0/0 BND EOR
%   B103:0/0  FAIL_OS  "Inspection Fail for Timed Logic" %
%   B103:14/15  BAREJECT16 %
%   B103:15/0  DAREJECT1 %
% Rung: 170 %
SOR XIC B103:15/0 BST TON T104:80 0.001 99 0 NXB XIC T104:80/DN BST OTU B103:15/0 NXB OTL B103:0/1 BND BND EOR
%   B103:15/0  DAREJECT1 %
%   B103:0/1  TIME2REJECT  "Timed Rejection Event" %
% Rung: 171 %
SOR XIC B103:0/0 XIC B103:15/0 XIO B103:15/1 BST OTL B103:15/1 NXB OTU B103:0/0 BND EOR
%   B103:0/0  FAIL_OS  "Inspection Fail for Timed Logic" %
%   B103:15/0  DAREJECT1 %
%   B103:15/1  DAREJECT2 %

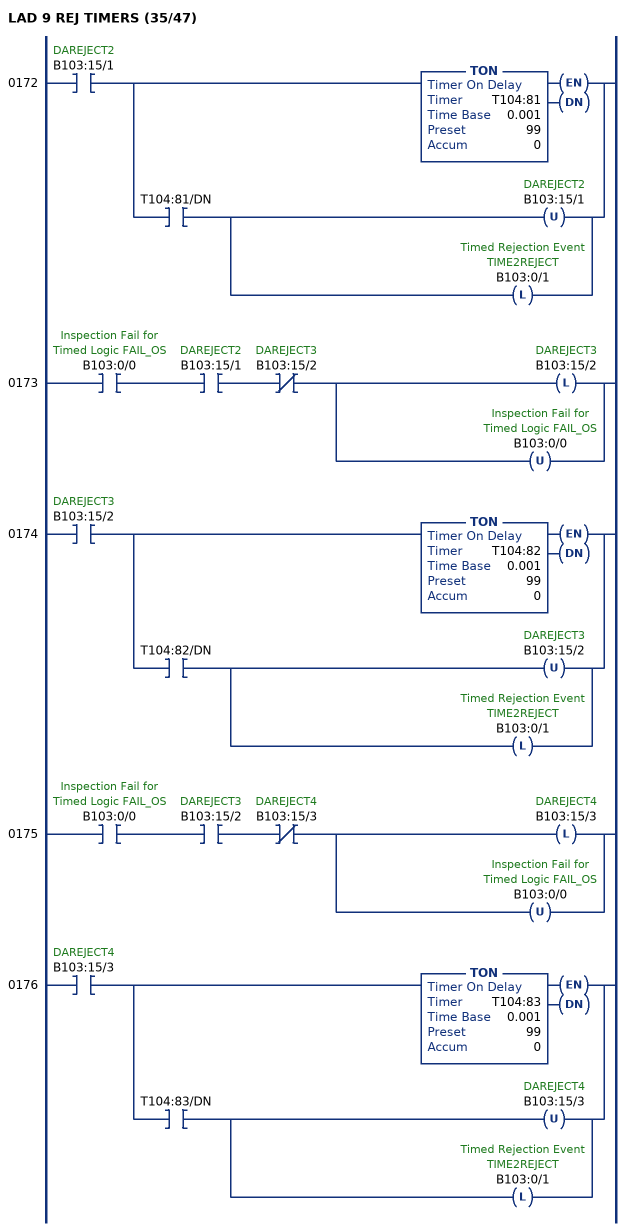
% Rung: 172 %
SOR XIC B103:15/1 BST TON T104:81 0.001 99 0 NXB XIC T104:81/DN BST OTU B103:15/1 NXB OTL B103:0/1 BND BND EOR
%   B103:15/1  DAREJECT2 %
%   B103:0/1  TIME2REJECT  "Timed Rejection Event" %
% Rung: 173 %
SOR XIC B103:0/0 XIC B103:15/1 XIO B103:15/2 BST OTL B103:15/2 NXB OTU B103:0/0 BND EOR
%   B103:0/0  FAIL_OS  "Inspection Fail for Timed Logic" %
%   B103:15/1  DAREJECT2 %
%   B103:15/2  DAREJECT3 %
% Rung: 174 %
SOR XIC B103:15/2 BST TON T104:82 0.001 99 0 NXB XIC T104:82/DN BST OTU B103:15/2 NXB OTL B103:0/1 BND BND EOR
%   B103:15/2  DAREJECT3 %
%   B103:0/1  TIME2REJECT  "Timed Rejection Event" %
% Rung: 175 %
SOR XIC B103:0/0 XIC B103:15/2 XIO B103:15/3 BST OTL B103:15/3 NXB OTU B103:0/0 BND EOR
%   B103:0/0  FAIL_OS  "Inspection Fail for Timed Logic" %
%   B103:15/2  DAREJECT3 %
%   B103:15/3  DAREJECT4 %
% Rung: 176 %
SOR XIC B103:15/3 BST TON T104:83 0.001 99 0 NXB XIC T104:83/DN BST OTU B103:15/3 NXB OTL B103:0/1 BND BND EOR
%   B103:15/3  DAREJECT4 %
%   B103:0/1  TIME2REJECT  "Timed Rejection Event" %

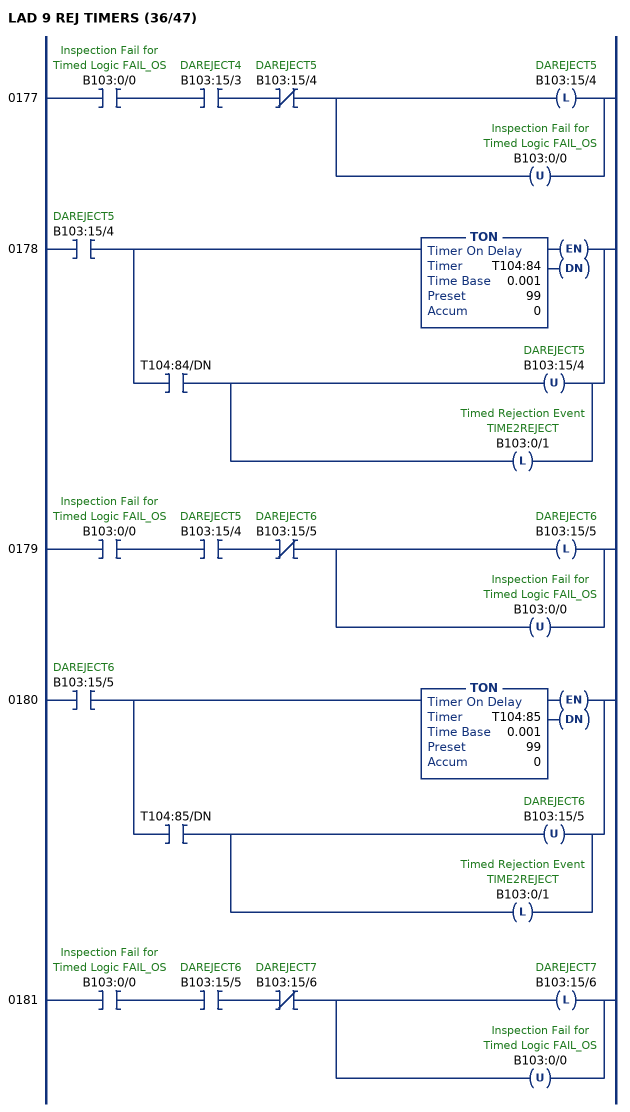
% Rung: 177 %
SOR XIC B103:0/0 XIC B103:15/3 XIO B103:15/4 BST OTL B103:15/4 NXB OTU B103:0/0 BND EOR
%   B103:0/0  FAIL_OS  "Inspection Fail for Timed Logic" %
%   B103:15/3  DAREJECT4 %
%   B103:15/4  DAREJECT5 %
% Rung: 178 %
SOR XIC B103:15/4 BST TON T104:84 0.001 99 0 NXB XIC T104:84/DN BST OTU B103:15/4 NXB OTL B103:0/1 BND BND EOR
%   B103:15/4  DAREJECT5 %
%   B103:0/1  TIME2REJECT  "Timed Rejection Event" %
% Rung: 179 %
SOR XIC B103:0/0 XIC B103:15/4 XIO B103:15/5 BST OTL B103:15/5 NXB OTU B103:0/0 BND EOR
%   B103:0/0  FAIL_OS  "Inspection Fail for Timed Logic" %
%   B103:15/4  DAREJECT5 %
%   B103:15/5  DAREJECT6 %
% Rung: 180 %
SOR XIC B103:15/5 BST TON T104:85 0.001 99 0 NXB XIC T104:85/DN BST OTU B103:15/5 NXB OTL B103:0/1 BND BND EOR
%   B103:15/5  DAREJECT6 %
%   B103:0/1  TIME2REJECT  "Timed Rejection Event" %
% Rung: 181 %
SOR XIC B103:0/0 XIC B103:15/5 XIO B103:15/6 BST OTL B103:15/6 NXB OTU B103:0/0 BND EOR
%   B103:0/0  FAIL_OS  "Inspection Fail for Timed Logic" %
%   B103:15/5  DAREJECT6 %
%   B103:15/6  DAREJECT7 %

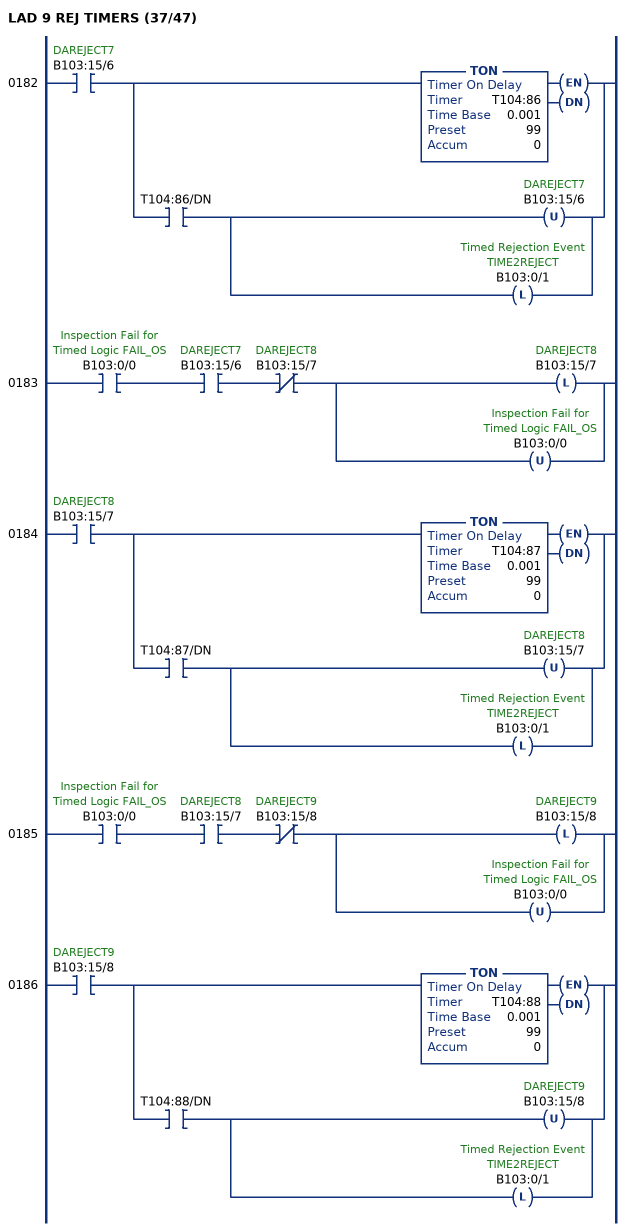
% Rung: 182 %
SOR XIC B103:15/6 BST TON T104:86 0.001 99 0 NXB XIC T104:86/DN BST OTU B103:15/6 NXB OTL B103:0/1 BND BND EOR
%   B103:15/6  DAREJECT7 %
%   B103:0/1  TIME2REJECT  "Timed Rejection Event" %
% Rung: 183 %
SOR XIC B103:0/0 XIC B103:15/6 XIO B103:15/7 BST OTL B103:15/7 NXB OTU B103:0/0 BND EOR
%   B103:0/0  FAIL_OS  "Inspection Fail for Timed Logic" %
%   B103:15/6  DAREJECT7 %
%   B103:15/7  DAREJECT8 %
% Rung: 184 %
SOR XIC B103:15/7 BST TON T104:87 0.001 99 0 NXB XIC T104:87/DN BST OTU B103:15/7 NXB OTL B103:0/1 BND BND EOR
%   B103:15/7  DAREJECT8 %
%   B103:0/1  TIME2REJECT  "Timed Rejection Event" %
% Rung: 185 %
SOR XIC B103:0/0 XIC B103:15/7 XIO B103:15/8 BST OTL B103:15/8 NXB OTU B103:0/0 BND EOR
%   B103:0/0  FAIL_OS  "Inspection Fail for Timed Logic" %
%   B103:15/7  DAREJECT8 %
%   B103:15/8  DAREJECT9 %
% Rung: 186 %
SOR XIC B103:15/8 BST TON T104:88 0.001 99 0 NXB XIC T104:88/DN BST OTU B103:15/8 NXB OTL B103:0/1 BND BND EOR
%   B103:15/8  DAREJECT9 %
%   B103:0/1  TIME2REJECT  "Timed Rejection Event" %

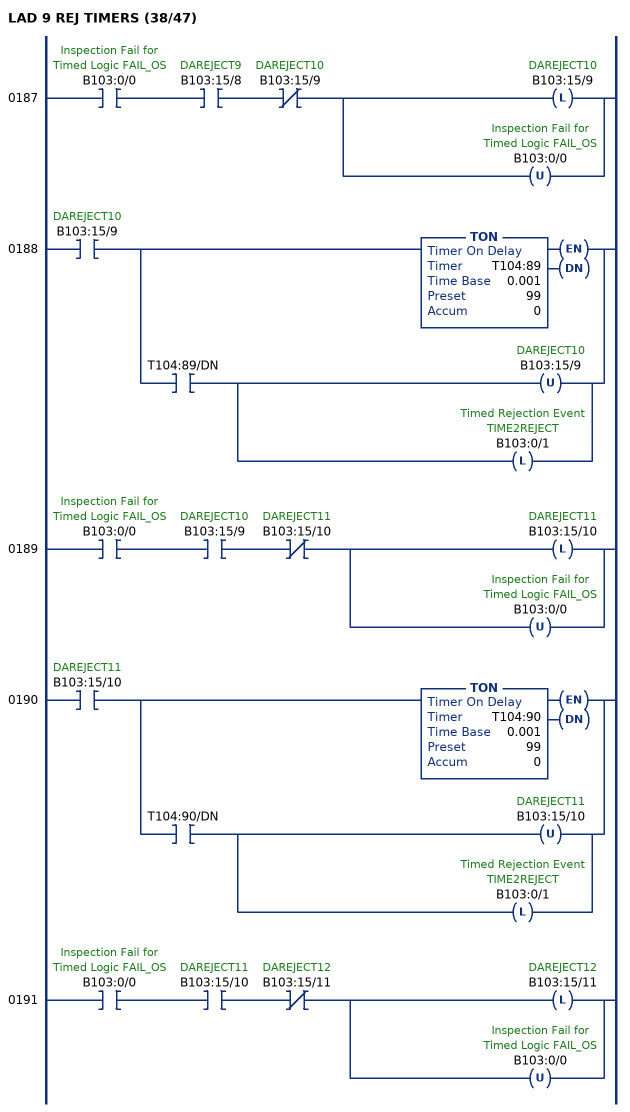
% Rung: 187 %
SOR XIC B103:0/0 XIC B103:15/8 XIO B103:15/9 BST OTL B103:15/9 NXB OTU B103:0/0 BND EOR
%   B103:0/0  FAIL_OS  "Inspection Fail for Timed Logic" %
%   B103:15/8  DAREJECT9 %
%   B103:15/9  DAREJECT10 %
% Rung: 188 %
SOR XIC B103:15/9 BST TON T104:89 0.001 99 0 NXB XIC T104:89/DN BST OTU B103:15/9 NXB OTL B103:0/1 BND BND EOR
%   B103:15/9  DAREJECT10 %
%   B103:0/1  TIME2REJECT  "Timed Rejection Event" %
% Rung: 189 %
SOR XIC B103:0/0 XIC B103:15/9 XIO B103:15/10 BST OTL B103:15/10 NXB OTU B103:0/0 BND EOR
%   B103:0/0  FAIL_OS  "Inspection Fail for Timed Logic" %
%   B103:15/9  DAREJECT10 %
%   B103:15/10  DAREJECT11 %
% Rung: 190 %
SOR XIC B103:15/10 BST TON T104:90 0.001 99 0 NXB XIC T104:90/DN BST OTU B103:15/10 NXB OTL B103:0/1 BND BND EOR
%   B103:15/10  DAREJECT11 %
%   B103:0/1  TIME2REJECT  "Timed Rejection Event" %
% Rung: 191 %
SOR XIC B103:0/0 XIC B103:15/10 XIO B103:15/11 BST OTL B103:15/11 NXB OTU B103:0/0 BND EOR
%   B103:0/0  FAIL_OS  "Inspection Fail for Timed Logic" %
%   B103:15/10  DAREJECT11 %
%   B103:15/11  DAREJECT12 %

